// TIA Portal project "test_web_CONECT_TCP_SERVER" (V15)

(* hardware
DEVICE "S7-1200 station_1"  S7-1200 Station
   slot 0: "Rack_0"  S7-1200 Rack  Rack  V1.0
   slot 1: "PLC_1"  CPU 1214C DC/DC/DC  6ES7 214-1AG40-0XB0  V4.2
*)

// ===== PLC "PLC_1"  CPU 1214C DC/DC/DC =====

VAR_GLOBAL   // PLC tag table "Default tag table"
   "System_Byte" AT %MB1 : Byte;
   "FirstScan" AT %M1.0 : Bool;
   "DiagStatusUpdate" AT %M1.1 : Bool;
   "AlwaysTRUE" AT %M1.2 : Bool;
   "AlwaysFALSE" AT %M1.3 : Bool;
   "Clock_Byte" AT %MB0 : Byte;
   "Clock_10Hz" AT %M0.0 : Bool;
   "Clock_5Hz" AT %M0.1 : Bool;
   "Clock_2.5Hz" AT %M0.2 : Bool;
   "Clock_2Hz" AT %M0.3 : Bool;
   "Clock_1.25Hz" AT %M0.4 : Bool;
   "Clock_1Hz" AT %M0.5 : Bool;
   "Clock_0.625Hz" AT %M0.6 : Bool;
   "Clock_0.5Hz" AT %M0.7 : Bool;
   "Tag_1" AT %MW0 : Int;
END_VAR

VAR_GLOBAL   // PLC tag table "output"
   "q0.4" AT %Q0.4 : Bool;
END_VAR

VAR_GLOBAL   // PLC tag table "hmi"
   "hmi_start_1" AT %M200.0 : Bool;
   "hmi_stop_1" AT %M200.1 : Bool;
   "hmi_dc_1" AT %Q0.5 : Bool;
END_VAR

DATA_BLOCK "web_com"   // DB1
{ S7_Optimized_Access := 'TRUE' }
VERSION : 0.1
   VAR
      tag_bool : Bool;
      tag_integer : Int;
      tag_byte : Byte;
      tag_real : Real;
      tag_string : String;
      tag_integer_2 : Int;
      Start : Bool;
      Stop : Bool;
      Data1 : Int;
      Data2 : Int;
   END_VAR
BEGIN
END_DATA_BLOCK

DATA_BLOCK "tcp_server"   // DB2
{ S7_Optimized_Access := 'TRUE' }
VERSION : 0.1
   VAR
      connect : TCON_IP_v4;
      NDR : Bool;
      DR : Bool;
      ERROR : Bool;
      STATUS : Word;
      DISCONECT : Bool;
   END_VAR
BEGIN
   connect.InterfaceId := 64;
   connect.ID := 1;
   connect.ConnectionType := 11;
   connect.RemoteAddress.ADDR[4] := 123;
   connect.RemoteAddress.ADDR[3] := 0;
   connect.RemoteAddress.ADDR[2] := 168;
   connect.RemoteAddress.ADDR[1] := 192;
   connect.LocalPort := 502;
END_DATA_BLOCK

DATA_BLOCK "data_tcp_server"   // DB3
{ S7_Optimized_Access := 'FALSE' }
VERSION : 0.1
   VAR
      holding_res : Array[0..20] of Int;
   END_VAR
BEGIN
END_DATA_BLOCK

FUNCTION "hmi" : Void   // FC1, LAD
{ S7_Optimized_Access := 'TRUE' }
VERSION : 0.1
BEGIN

REGION Network 1
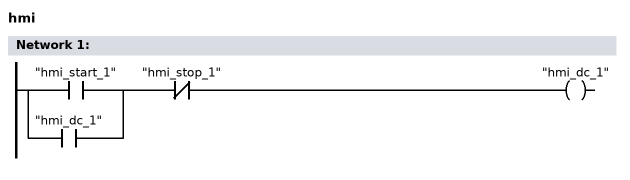
   RUNG wire#powerrail
      Contact( "hmi_start_1" )
      wire#w1
      I_Contact( "hmi_stop_1" )
      Coil( "hmi_dc_1" )
   END_RUNG
   RUNG wire#powerrail
      Contact( "hmi_dc_1" )
   END_RUNG wire#w1
   // the same network as SCL:
   "hmi_dc_1" := ("hmi_start_1" OR "hmi_dc_1") AND NOT "hmi_stop_1";
END_REGION
END_FUNCTION

ORGANIZATION_BLOCK "Main"   // OB1, LAD, ProgramCycle
TITLE = "Main Program Sweep (Cycle)"
{ S7_Optimized_Access := 'TRUE' }
VERSION : 0.1
   VAR_INPUT
      Initial_Call : Bool;   // Initial call of this OB
      Remanence : Bool;   // =True, if remanent data are available
   END_VAR
BEGIN

REGION Network 1
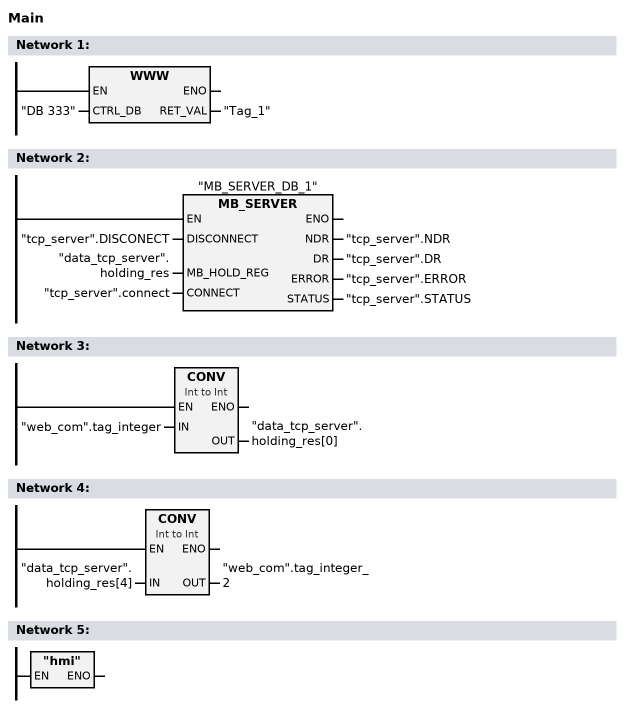
   "Tag_1" := WWW(CTRL_DB := "DB 333");
END_REGION

REGION Network 2
   "MB_SERVER_DB_1"(DISCONNECT := "tcp_server".DISCONECT,   // MB_SERVER
                    MB_HOLD_REG := "data_tcp_server".holding_res,
                    CONNECT := "tcp_server".connect,
                    NDR => "tcp_server".NDR,
                    DR => "tcp_server".DR,
                    ERROR => "tcp_server".ERROR,
                    STATUS => "tcp_server".STATUS);
END_REGION

REGION Network 3
   RUNG wire#powerrail
      { S7_Templates := "[SrcType := Int, DestType := Int]" } Convert(in := "web_com".tag_integer, out => "data_tcp_server".holding_res[0])
   END_RUNG
   // the same network as SCL:
   "data_tcp_server".holding_res[0] := INT_TO_INT("web_com".tag_integer);
END_REGION

REGION Network 4
   RUNG wire#powerrail
      { S7_Templates := "[SrcType := Int, DestType := Int]" } Convert(in := "data_tcp_server".holding_res[4], out => "web_com".tag_integer_2)
   END_RUNG
   // the same network as SCL:
   "web_com".tag_integer_2 := INT_TO_INT("data_tcp_server".holding_res[4]);
END_REGION

REGION Network 5
   RUNG wire#powerrail
      "hmi"()
   END_RUNG
   // the same network as SCL:
   "hmi"();
END_REGION
END_ORGANIZATION_BLOCK